FUNCTION_BLOCK E_PULSE_RETRIG (* standard timer function block (pulse) - retriggerable version *)
  (* Standard: 61499-2; Description: Copyright (c) 2023 HR Agrartechnik GmbH This program and the accompanying materials are made available under the terms of the Eclipse Public License 2.0 which is available at https://www.eclipse.org/legal/epl-2.0/ SPDX-License-Identifier: EPL-2.0 E_TP -- Impulse forming FB (Retriggerable) Generate a Impulse with a given Time. This FB makes a Impulse of Duration TM on the Output QO. New REQ restarts the timer. *)
  (* Version 1.1, 2026-04-19, Franz Höpfinger, HR Agrartechnik GmbH, retriggerable version *)
  (* Version 3.0, 2025-04-14, Patrick Aigner, changed package *)
  (* Version 1.1, 2024-04-23, Franz Höpfinger, HR Agrartechnik GmbH, Add a Reset to Timer FBs *)
  (* Version 1.0.1, 2024-03-05, Franz Höpfinger, HR Agrartechnik GmbH, renamed to E_PULSE *)
  (* Version 1.0, 2023-08-21, Franz Höpfinger, HR Agrartechnik GmbH, initial implementation as E_IMPULSE *)
  PACKAGE iec61499::events::timers;
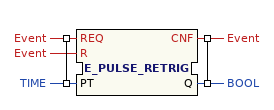
  EVENT_INPUT
    REQ WITH PT; (* Service Request (Restarts the timer) *)
    R; (* Reset *)
  END_EVENT
  EVENT_OUTPUT
    CNF WITH Q; (* Confirmation of Requested Service *)
  END_EVENT
  VAR_INPUT
    PT : TIME; (* Pulse time *)
  END_VAR
  VAR_OUTPUT
    Q : BOOL; (* Output *)
  END_VAR
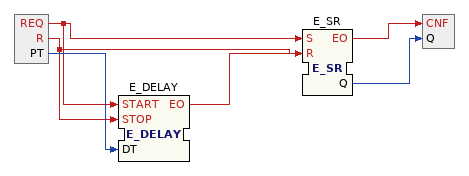
  FBS
    E_DELAY : iec61499::events::E_DELAY;
    E_SR : iec61499::events::E_SR;
  END_FBS
  EVENT_CONNECTIONS
    REQ TO E_DELAY.START;
    REQ TO E_SR.S;
    E_DELAY.EO TO E_SR.R;
    E_SR.EO TO CNF;
    R TO E_DELAY.STOP;
    R TO E_SR.R;
  END_CONNECTIONS
  DATA_CONNECTIONS
    PT TO E_DELAY.DT;
    E_SR.Q TO Q;
  END_CONNECTIONS
END_FUNCTION_BLOCK
